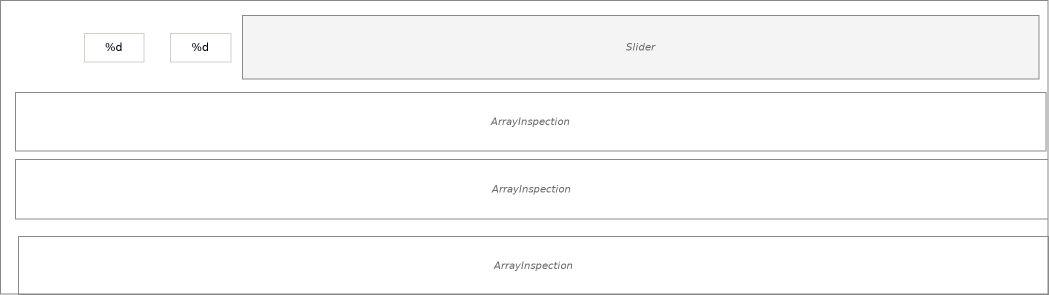
VISUALIZATION SorterArray  // 1049x295
    Frame (15,92 1031x59)
        shows ArrayInspection(st_ItemExt_Disp := MAIN.st_DisplayItem)
        shows ArrayInspection()
        shows ArrayInspection()
    Textfield (170,33 61x29), "%d", text variable: MAIN.nDisplayItemIndex
        OnMouseDown: write MAIN.nDisplayItemIndex via Edit
    Slider (242,15 797x64), variable: MAIN.nDisplayItemIndex, scale 0..100
    Textfield (84,33 60x29), "%d", text variable: MAIN.st_SorterEncoder.CurrentCount
    Frame (15,159 1033x60)
        shows ArrayInspection(st_ItemExt_Disp := ProcessBuffers_P2140.st_DisplayItem)
    Frame (18,236 1031x59)
        shows ArrayInspection(st_ItemExt_Disp := Sorter_P2140.st_DisplayItem)
END_VISUALIZATION

(* stored: Version 1.1.0.1, ProductVersion 3.1.4024.4
   Visu SorterArray: Id {1234879f-8573-4a83-802b-e47f6cefc207} *)
